//=============================================================================
// ST_HmiSetpoints
//-----------------------------------------------------------------------------
// Direction: Pi -> PLC (request) and PLC -> Pi (applied echo in ST_HmiStatus).
// Pi writes the whole struct, then pulses stCommand.bApplySetpoints.
// FB_Hmi clamps each value to ST_SetpointLimits before applying, and the
// clamped result is echoed in ST_HmiStatus.rSet*Applied so the UI always
// shows the truth, not the request.
//=============================================================================
{attribute 'pack_mode' := '1'}
TYPE ST_HmiSetpoints :
STRUCT
	bSetPurgeOnStartup	: BOOL := FALSE;	// 
	rSetFlow       		: REAL;  			// requested flow setpoint      [SLM]
    //rSetDsPressure 		: REAL; 			// downstream pressure setpoint [Torr]
	rSetElevation		: REAL;				// meters above seal level [MASL] 
	bSetSize25L			: BOOL;				// set size to 25L, FALSE = 50L
	sSetEipAddress		: STRING(15);		// string to represent EthernetIP address
END_STRUCT
END_TYPE

(* stored: Version 1.1.0.1, ProductVersion 3.1.4026.19
   DUT ST_HmiSetpoints: Id {a1b2c3d4-0006-4a5b-9c8d-e1f200000006} *)
